(*======================================================================================================================================*)
(*fb_timeDiffLite:	Neuer einfacherer Baustein, welcher nur über Start funktioniert *)
(*
Date          	| Version    	| created under        	| Author          	| Remark *)
(*======================================================================================================================================*)
(*03/09/2025   	| 1.00      	| TC3		  			| N.Kersting       | first release *)
(*======================================================================================================================================*)
FUNCTION_BLOCK fb_timeDiffLite_libversion
VAR_INPUT
	I_bStart	:BOOL;
	I_bReset	:BOOL;
END_VAR
VAR_OUTPUT
	Q_tDiffTime	:TIME;
END_VAR
VAR
	tStart	:TIME;
	tStop	:TIME;

	rTrigStart:	R_TRIG;
	rTrigStop:	R_TRIG;
	bMem: BOOL;
END_VAR

rTrigStart(CLK:=I_bStart);

IF	I_bReset	
THEN	
	bMem := FALSE;
	tStart:= T#0S;
	tStop:=T#0S;
ELSE
	
	IF	rTrigStart.Q	
		AND bMem
	THEN	
		bMem := FALSE; 
		tStart:= TIME();
		Q_tDiffTime:=	tStart-tStop;
	END_IF

	IF	rTrigStart.Q
		AND NOT bMem	
	THEN	
		bMem := TRUE;
		tStop:=	TIME();
	END_IF
END_IF

END_FUNCTION_BLOCK

(* stored: Version 1.1.0.1, ProductVersion 3.1.4024.15
   POU fb_timeDiffLite_libversion: Id {c07171d1-5f86-476d-b836-6c646ec75bde}, SpecialFunc None *)
